// TwinCAT 3 PLC project Haltbergholz
// ProgramVersion: 3.1.4026.19
// libraries:
//   Tc2_ModbusSrv, * (Beckhoff Automation GmbH)
//   Tc2_Standard, * (Beckhoff Automation GmbH)
//   Tc2_System, * (Beckhoff Automation GmbH)
//   Tc2_Utilities, * (Beckhoff Automation GmbH)
//   Tc3_EventLogger, * (Beckhoff Automation GmbH)
// project tree:
//   DUTs/ E_PhaseSelect.TcDUT, E_StorageChargeState.TcDUT
//   DUTs/FroniusModbusRegisterMapping/ ST_RegMapInverter.TcDUT, ST_RegMapMeter.TcDUT, ST_RegMapStorage.TcDUT
//   DUTs/GridOperatingData/ ST_OpDataInverter.TcDUT, ST_OpDataMeter.TcDUT, ST_OpDataStorage.TcDUT
//   DUTs/LoadControlData/ ST_CtrlDataPower.TcDUT, ST_CtrlDataSetpoint.TcDUT
//   DUTs/Properties/ ST_SchmittTriggerProperties.TcDUT
//   / PlcTask.TcTTO
//   POUs/ FB_ModbusCon.TcPOU, FB_SchmittTrigger.TcPOU, F_MovingAverage.TcPOU, I_LoadCtrl.TcIO, MainCtrl.TcPOU
// real-time tasks:
//   TASK PlcTask: cycle T#10ms, priority 20, ADS port 350

CONFIGURATION Haltbergholz
    RESOURCE PLC ON TwinCAT3
        TASK PlcTask(INTERVAL := T#10ms, PRIORITY := 20);
        PROGRAM MainCtrl WITH PlcTask : MainCtrl;
    END_RESOURCE
END_CONFIGURATION

// ---- DUTs/E_PhaseSelect.TcDUT
{attribute 'qualified_only'}
{attribute 'strict'}
{attribute 'to_string'}
TYPE E_PhaseSelect :
(
	ALL := 0,
    L1,
    L2,
    L3
);
END_TYPE

// ---- DUTs/E_StorageChargeState.TcDUT
{attribute 'qualified_only'}
{attribute 'strict'}
{attribute 'to_string'}
TYPE E_StorageChargeState :
(
	off := 1,
    empty := 2,
    discharging := 3,
    charging := 4,
    full := 5,
    holding := 6,
    testing := 7
) WORD;
END_TYPE

// ---- DUTs/FroniusModbusRegisterMapping/ST_RegMapInverter.TcDUT
TYPE ST_RegMapInverter :
STRUCT
    // Register 40072
    nCurrentTotal: WORD;
    // Register 40073
    nCurrentL1: WORD;
    // Register 40074
    nCurrentL2: WORD;
    // Register 40075
    nCurrentL3: WORD;
    // Register 40076
    nSfCurrent: WORD;
    // Register 40077
    nVoltageL1L2: WORD;
    // Register 40078
    nVoltageL2L3: WORD;
    // Register 40079
    nVoltageL3L1: WORD;
    // Register 40080
    nVoltageL1N: WORD;
    // Register 40081
    nVoltageL2N: WORD;
    // Register 40082
    nVoltageL3N: WORD;
    // Register 40083
    nSfVoltage: WORD;
    // Register 40084
    nPower: WORD;
    // Register 40085
    nSfPower: WORD;
    // Register 40086
    nFrequency: WORD;
    // Register 40087
    nSfFrequency: WORD;
END_STRUCT
END_TYPE

// ---- DUTs/FroniusModbusRegisterMapping/ST_RegMapMeter.TcDUT
TYPE ST_RegMapMeter :
STRUCT
    // Register 40072
    nCurrentTotal: WORD;
    // Register 40073
    nCurrentL1: WORD;
    // Register 40074
    nCurrentL2: WORD;
    // Register 40075
    nCurrentL3: WORD;
    // Register 40076
    nSfCurrent: WORD;
    // Register 40077
    nVoltageLN: WORD;
    // Register 40078
    nVoltageL1N: WORD;
    // Register 40079
    nVoltageL2N: WORD;
    // Register 40080
    nVoltageL3N: WORD;
    // Register 40081
    nVoltageLL: WORD;
    // Register 40082
    nVoltageL1L2: WORD;
    // Register 40083
    nVoltageL2L3: WORD;
    // Register 40084
    nVoltageL3L1: WORD;
    // Register 40085
    nSfVoltage: WORD;
    // Register 40086
    nFrequency: WORD;
    // Register 40087
    nSfFrequency: WORD;
    // Register 40088
    nPower: WORD;
    // Register 40089
    nPowerL1: WORD;
    // Register 40090
    nPowerL2: WORD;
    // Register 40091
    nPowerL3: WORD;
    // Register 40092
    nSfPower: WORD;
END_STRUCT
END_TYPE

// ---- DUTs/FroniusModbusRegisterMapping/ST_RegMapStorage.TcDUT
TYPE ST_RegMapStorage :
STRUCT
    // Register 40352
    nStateOfCharge: WORD;
    // Register 40353
    nStorageAvailable: WORD;
    // Register 40354
    nVoltageInternal: WORD;
    // Register 40355
    nState: E_StorageChargeState;
    // Register 40366, fixed to -2
    nSfStateOfCharge: WORD := INT_TO_UINT(-2);
END_STRUCT
END_TYPE

// ---- DUTs/GridOperatingData/ST_OpDataInverter.TcDUT
TYPE ST_OpDataInverter :
STRUCT
    // Operating data refreshed in this cycle
    bOpDataIsUpdated: BOOL;
    // Current Phase L1 [A]
    fCurrentL1: REAL;
    // Current Phase L2 [A]
    fCurrentL2: REAL;
    // Current Phase L3 [A]
    fCurrentL3: REAL;
    // Voltage between Phase L1 and L2 [V]
    fVoltageL1L2: REAL;
    // Voltage between Phase L2 and L3 [V]
    fVoltageL2L3: REAL;
    // Voltage between Phase L3 and L1 [V]
    fVoltageL3L1: REAL;
    // Voltage between Phase L1 and N [V]
    fVoltageL1N: REAL;
    // Voltage between Phase L2 and N [V]
    fVoltageL2N: REAL;
    // Voltage between Phase L3 and N [V]
    fVoltageL3N: REAL;
    // Total Real Power [W]
    fPower: REAL;
    // Frequency [Hz]
    fFrequency: REAL;
END_STRUCT
END_TYPE

// ---- DUTs/GridOperatingData/ST_OpDataMeter.TcDUT
TYPE ST_OpDataMeter :
STRUCT
    // Operating data refreshed in this cycle
    bOpDataIsUpdated: BOOL;
    // Current Phase L1 [A]
    fCurrentL1: REAL;
    // Current Phase L2 [A]
    fCurrentL2: REAL;
    // Current Phase L3 [A]
    fCurrentL3: REAL;
    // Voltage between Phase L1 and L2 [V]
    fVoltageL1L2: REAL;
    // Voltage between Phase L2 and L3 [V]
    fVoltageL2L3: REAL;
    // Voltage between Phase L3 and L1 [V]
    fVoltageL3L1: REAL;
    // Voltage between Phase L1 and N [V]
    fVoltageL1N: REAL;
    // Voltage between Phase L2 and N [V]
    fVoltageL2N: REAL;
    // Voltage between Phase L3 and N [V]
    fVoltageL3N: REAL;
    // Total Real Power [W]
    fPower: REAL;
    // Real Power of Phase L1 [W]
    fPowerL1: REAL;
    // Real Power of Phase L2 [W]
    fPowerL2: REAL;
    // Real Power of Phase L3 [W]
    fPowerL3: REAL;
    // Frequency [Hz]
    fFrequency: REAL;
END_STRUCT
END_TYPE

// ---- DUTs/GridOperatingData/ST_OpDataStorage.TcDUT
TYPE ST_OpDataStorage :
STRUCT
    // Operating data refreshed in this cycle
    bOpDataIsUpdated: BOOL;
    // Currently available energy as a percent of the capacity rating
    nStateOfCharge: INT;
    // Charge status of storage device
    eState: E_StorageChargeState;
END_STRUCT
END_TYPE

// ---- DUTs/LoadControlData/ST_CtrlDataPower.TcDUT
TYPE ST_CtrlDataPower :
STRUCT
    // Real Power of Phase L1 [W]
    fPowerL1: REAL;
    // Real Power of Phase L2 [W]
    fPowerL2: REAL;
    // Real Power of Phase L3 [W]
    fPowerL3: REAL;
END_STRUCT
END_TYPE

// ---- DUTs/LoadControlData/ST_CtrlDataSetpoint.TcDUT
TYPE ST_CtrlDataSetpoint :
STRUCT
    // Load setpoint for Phase L1 [0-255]
    nLoadSetpointL1: USINT;
    // Load setpoint for Phase L2 [0-255]
    nLoadSetpointL2: USINT;
    // Load setpoint for Phase L3 [0-255]
    nLoadSetpointL3: USINT;
END_STRUCT
END_TYPE

// ---- DUTs/Properties/ST_SchmittTriggerProperties.TcDUT
TYPE ST_SchmittTriggerProperties :
STRUCT
    // Number of oscillations (t < threashold) required to reverse output
    nLimitOscillations: INT;
    // Time threshold to switch output after falling edge of input
    tFallThreshold: TIME;
    // Time threshold to switch output after rising edge of input
    tRiseThreshold: TIME;
END_STRUCT
END_TYPE

// ---- POUs/I_LoadCtrl.TcIO
INTERFACE I_LoadCtrl

// True if load is ready to powered on
{attribute 'monitoring' := 'variable'}
PROPERTY bReady : BOOL
GET
END_GET
END_PROPERTY

// Show only events with minimum severety level
{attribute 'monitoring' := 'call'}
PROPERTY eTraceLevel: Global.TcEventSeverity
GET
END_GET
SET
END_SET
END_PROPERTY

// Release power up of load on selected phase
METHOD PowerDown : BOOL
VAR_INPUT
    ePhase: E_PhaseSelect := E_PhaseSelect.ALL;
END_VAR
END_METHOD

// Power down load on selected phase
METHOD PowerUp : BOOL
VAR_INPUT
    ePhase: E_PhaseSelect := E_PhaseSelect.ALL;
END_VAR
END_METHOD

// Request setpoint for poweroutput relative to stPowerMaximum
{attribute 'monitoring' := 'call'}
PROPERTY stLoadSetpoint : REFERENCE TO ST_CtrlDataSetpoint
GET
END_GET
SET
END_SET
END_PROPERTY

// Actual power used from load
{attribute 'monitoring' := 'variable'}
PROPERTY stPowerActual : REFERENCE TO ST_CtrlDataPower
GET
END_GET
END_PROPERTY

// Minimum power on lowest setpoint
{attribute 'monitoring' := 'variable'}
PROPERTY stPowerMaximum : REFERENCE TO ST_CtrlDataPower
GET
END_GET
END_PROPERTY

// Maxmimum power on highest setpoint
{attribute 'monitoring' := 'variable'}
PROPERTY stPowerMinimum : REFERENCE TO ST_CtrlDataPower
GET
END_GET
END_PROPERTY

END_INTERFACE

// ---- POUs/MainCtrl.TcPOU
PROGRAM MainCtrl
VAR
    fbReadOpData: FB_ModbusCon := (
                    sInverterIPAddr := '127.0.0.1',
                    nInverterTCPPort := 5502,
                    nInverterUnitID := 16#01,
                    nMeterUnitID := 16#C8,
                    tConnectionTimeout := T#10S,
                    tConnectionCoolDown := T#10S);

    // Load control 1
    ipLoad1: I_LoadCtrl;

    // Battery is charging
    fbStorageIsCharging: FB_SchmittTrigger;

    // Temporary Power of Phase L1 values used for moving average 
    aMeterHistoryPowerL1: ARRAY[1..nSamplesMovingAverage] OF REAL;
    nMeterHistoryCursorPowerL1: INT;
    // Temporary Power of Phase L2 values used for moving average 
    aMeterHistoryPowerL2: ARRAY[1..nSamplesMovingAverage] OF REAL;
    nMeterHistoryCursorPowerL2: INT;
    // Temporary Power of Phase L3 values used for moving average 
    aMeterHistoryPowerL3: ARRAY[1..nSamplesMovingAverage] OF REAL;
    nMeterHistoryCursorPowerL3: INT;

    // Actual power feed to grid (>0: feed to grid, <0: draw from grid)
    stSurplusPower: ST_CtrlDataPower;
    // Surplus available at Phase L1
    fbSurplusAvailableL1: FB_SchmittTrigger;
    // Surplus available at Phase L2
    fbSurplusAvailableL2: FB_SchmittTrigger;
    // Surplus available at Phase L3
    fbSurplusAvailableL3: FB_SchmittTrigger;
END_VAR
VAR PERSISTENT
    // Battery state of charge is high
    nStorageStateOfChargeHigh: INT := 75;
    // Schmitt trigger configuration for battery charging state while battery state of charge low
    stStorageIsChargingTriggerPropertiesLow: ST_SchmittTriggerProperties := (
                                        nLimitOscillations := 3,
                                        tFallThreshold := T#5M,
                                        tRiseThreshold := T#2M);
    // Schmitt trigger configuration for battery charging state while battery state of charge high
    stStorageIsChargingTriggerPropertiesHigh: ST_SchmittTriggerProperties := (
                                        nLimitOscillations := 3,
                                        tFallThreshold := T#2M,
                                        tRiseThreshold := T#2M);
    // Schmitt trigger configuration for surplus power active while battery state of charge low
    stSurplusPowerTriggerPropertiesLow: ST_SchmittTriggerProperties := (
                                        nLimitOscillations := 3,
                                        tFallThreshold := T#5M,
                                        tRiseThreshold := T#1M);
    // Schmitt trigger configuration for surplus power active while battery state of charge high
    stSurplusPowerTriggerPropertiesHigh: ST_SchmittTriggerProperties := (
                                        nLimitOscillations := 3,
                                        tFallThreshold := T#50M,
                                        tRiseThreshold := T#1M);
    // Minimum amount of power feed to grid must be exceeded to show as surplus (>=0W)
    stSurplusPowerMinimum: ST_CtrlDataPower := (
                                        fPowerL1 := 20,
                                        fPowerL2 := 20,
                                        fPowerL3 := 20);
END_VAR
VAR CONSTANT
    // Number of samples for moving average calculation
    nSamplesMovingAverage: INT := 3;
END_VAR

// Fetch measurement data
fbReadOpData();

IF NOT fbReadOpData.bReady THEN
    fbReadOpData.bEnable := FALSE;
    RETURN;
ELSE
    fbReadOpData.bEnable := TRUE;
END_IF

// Battery measurement data is updated
IF fbReadOpData.stStorage.bOpDataIsUpdated THEN
    IF fbReadOpData.stStorage.nStateOfCharge > nStorageStateOfChargeHigh THEN
        fbStorageIsCharging.nLimitOscillations := stStorageIsChargingTriggerPropertiesLow.nLimitOscillations;
        fbStorageIsCharging.tFallThreshold := stStorageIsChargingTriggerPropertiesLow.tFallThreshold;
        fbStorageIsCharging.tRiseThreshold := stStorageIsChargingTriggerPropertiesLow.tRiseThreshold;
    ELSE
        fbStorageIsCharging.nLimitOscillations := stStorageIsChargingTriggerPropertiesHigh.nLimitOscillations;
        fbStorageIsCharging.tFallThreshold := stStorageIsChargingTriggerPropertiesHigh.tFallThreshold;
        fbStorageIsCharging.tRiseThreshold := stStorageIsChargingTriggerPropertiesHigh.tRiseThreshold;
    END_IF

    // Detect change on battery charging state
    fbStorageIsCharging.bIn := fbReadOpData.stStorage.eState = E_StorageChargeState.charging;
END_IF

fbStorageIsCharging();

// Meter measurement data is updated
IF fbReadOpData.stMeter.bOpDataIsUpdated THEN
    // Get moving average of power measured at meter and reverse sign (>0: feed to grid, <0: draw from grid)
    stSurplusPower.fPowerL1 := F_MovingAverage(fIn := fbReadOpData.stMeter.fPowerL1, aHisotry := aMeterHistoryPowerL1, nCursor := nMeterHistoryCursorPowerL1) * -1;
    stSurplusPower.fPowerL2 := F_MovingAverage(fIn := fbReadOpData.stMeter.fPowerL2, aHisotry := aMeterHistoryPowerL2, nCursor := nMeterHistoryCursorPowerL2) * -1;
    stSurplusPower.fPowerL3 := F_MovingAverage(fIn := fbReadOpData.stMeter.fPowerL3, aHisotry := aMeterHistoryPowerL3, nCursor := nMeterHistoryCursorPowerL3) * -1;

    // Add the actual power used of the loads to surplus (further calculations without used power of all load)
    IncludeLoadToSurplus(ipLoad := ipLoad1);

    // Generate setpoint for each load
    GenerateSetpoint(ipLoad := ipLoad1);

    // Detect change between power feed and draw to grid
    fbSurplusAvailableL1.bIn := stSurplusPower.fPowerL1 >= stSurplusPowerMinimum.fPowerL1;
    fbSurplusAvailableL2.bIn := stSurplusPower.fPowerL2 >= stSurplusPowerMinimum.fPowerL2;
    fbSurplusAvailableL3.bIn := stSurplusPower.fPowerL3 >= stSurplusPowerMinimum.fPowerL3;
END_IF

// Set properties of surplus available trigger based on battery charging state
IF fbStorageIsCharging.bOut THEN
    fbSurplusAvailableL1.nLimitOscillations := stSurplusPowerTriggerPropertiesLow.nLimitOscillations;
    fbSurplusAvailableL1.tFallThreshold := stSurplusPowerTriggerPropertiesLow.tFallThreshold;
    fbSurplusAvailableL1.tRiseThreshold := stSurplusPowerTriggerPropertiesLow.tRiseThreshold;
    fbSurplusAvailableL2.nLimitOscillations := stSurplusPowerTriggerPropertiesLow.nLimitOscillations;
    fbSurplusAvailableL2.tFallThreshold := stSurplusPowerTriggerPropertiesLow.tFallThreshold;
    fbSurplusAvailableL2.tRiseThreshold := stSurplusPowerTriggerPropertiesLow.tRiseThreshold;
    fbSurplusAvailableL3.nLimitOscillations := stSurplusPowerTriggerPropertiesLow.nLimitOscillations;
    fbSurplusAvailableL3.tFallThreshold := stSurplusPowerTriggerPropertiesLow.tFallThreshold;
    fbSurplusAvailableL3.tRiseThreshold := stSurplusPowerTriggerPropertiesLow.tRiseThreshold;
ELSE
    fbSurplusAvailableL1.nLimitOscillations := stSurplusPowerTriggerPropertiesHigh.nLimitOscillations;
    fbSurplusAvailableL1.tFallThreshold := stSurplusPowerTriggerPropertiesHigh.tFallThreshold;
    fbSurplusAvailableL1.tRiseThreshold := stSurplusPowerTriggerPropertiesHigh.tRiseThreshold;
    fbSurplusAvailableL2.nLimitOscillations := stSurplusPowerTriggerPropertiesHigh.nLimitOscillations;
    fbSurplusAvailableL2.tFallThreshold := stSurplusPowerTriggerPropertiesHigh.tFallThreshold;
    fbSurplusAvailableL2.tRiseThreshold := stSurplusPowerTriggerPropertiesHigh.tRiseThreshold;
    fbSurplusAvailableL3.nLimitOscillations := stSurplusPowerTriggerPropertiesHigh.nLimitOscillations;
    fbSurplusAvailableL3.tFallThreshold := stSurplusPowerTriggerPropertiesHigh.tFallThreshold;
    fbSurplusAvailableL3.tRiseThreshold := stSurplusPowerTriggerPropertiesHigh.tRiseThreshold;
END_IF

fbSurplusAvailableL1();
fbSurplusAvailableL2();
fbSurplusAvailableL3();

// Enable / Disable Load 1 on phase 1
IF fbSurplusAvailableL1.bOut AND ipLoad1.bReady THEN
    ipLoad1.PowerUp(ePhase := E_PhaseSelect.L1);
ELSE
    ipLoad1.PowerDown(ePhase := E_PhaseSelect.L1);
END_IF

// Enable / Disable Load 1 on phase 2
IF fbSurplusAvailableL2.bOut AND ipLoad1.bReady THEN
    ipLoad1.PowerUp(ePhase := E_PhaseSelect.L2);
ELSE
    ipLoad1.PowerDown(ePhase := E_PhaseSelect.L2);
END_IF

// Enable / Disable Load 1 on phase 3
IF fbSurplusAvailableL3.bOut AND ipLoad1.bReady THEN
    ipLoad1.PowerUp(ePhase := E_PhaseSelect.L3);
ELSE
    ipLoad1.PowerDown(ePhase := E_PhaseSelect.L3);
END_IF

// Generate and append setpoint of each phase to stLoadSetpoint of interface based on stPowerMaximum of interface and the current stSurplusPower 
METHOD PRIVATE GenerateSetpoint
VAR_INPUT
    // Interface of load control
    ipLoad: REFERENCE TO I_LoadCtrl;
END_VAR
IF ipLoad.stPowerMaximum.fPowerL1 <= 0 THEN
    ipLoad.stLoadSetpoint.nLoadSetpointL1 := 0;
ELSE
    ipLoad.stLoadSetpoint.nLoadSetpointL1 := REAL_TO_USINT(LIMIT(0, stSurplusPower.fPowerL1 / ipLoad.stPowerMaximum.fPowerL1, 1) * 255);
END_IF

IF ipLoad.stPowerMaximum.fPowerL2 <= 0 THEN
    ipLoad.stLoadSetpoint.nLoadSetpointL2 := 0;
ELSE
    ipLoad.stLoadSetpoint.nLoadSetpointL2 := REAL_TO_USINT(LIMIT(0, stSurplusPower.fPowerL2 / ipLoad.stPowerMaximum.fPowerL2, 1) * 255);
END_IF

IF ipLoad.stPowerMaximum.fPowerL3 <= 0 THEN
    ipLoad.stLoadSetpoint.nLoadSetpointL3 := 0;
ELSE
    ipLoad.stLoadSetpoint.nLoadSetpointL3 := REAL_TO_USINT(LIMIT(0, stSurplusPower.fPowerL3 / ipLoad.stPowerMaximum.fPowerL3, 1) * 255);
END_IF
END_METHOD

// Add the actual power used of the load to surplus
METHOD PRIVATE IncludeLoadToSurplus
VAR_INPUT
    // Interface of load control
    ipLoad: REFERENCE TO I_LoadCtrl;
END_VAR
stSurplusPower.fPowerL1 := stSurplusPower.fPowerL1 + ipLoad.stPowerActual.fPowerL1;
stSurplusPower.fPowerL2 := stSurplusPower.fPowerL2 + ipLoad.stPowerActual.fPowerL2;
stSurplusPower.fPowerL3 := stSurplusPower.fPowerL3 + ipLoad.stPowerActual.fPowerL3;
END_METHOD

END_PROGRAM

// ---- POUs/FB_ModbusCon.TcPOU
FUNCTION_BLOCK FB_ModbusCon
VAR_INPUT
    bEnable: BOOL;
END_VAR
VAR_OUTPUT
    // Operating data from inverter
    stInverter: ST_OpDataInverter;
    // Operating data from meter
    stMeter: ST_OpDataMeter;
    // Operating data from storage
    stStorage: ST_OpDataStorage;
    // Connection is ready and not locked out
    bReady: BOOL;
END_VAR
VAR
    // IP address of the target device
    {attribute 'hide'}
    _sInverterIPAddr: STRING;
    // Port number of the target device
    {attribute 'hide'}
    _nInverterTCPPort: UINT;
    // Modbus RTU ID of inverter, value must be 16#FF if addressed directly via TCP/IP
    {attribute 'hide'}
    _nInverterUnitID: BYTE;
    // Modbus RTU ID of meter, value must be 16#FF if addressed directly via TCP/IP
    {attribute 'hide'}
    _nMeterUnitID: BYTE;
    // Timeout that may not be exceeded by execution of the ADS command
    {attribute 'hide'}
    _tConnectionTimeout: TIME;
    // Timeout between modbus commands sent to target device
    {attribute 'hide'}
    _tConnectionCoolDown: TIME;

    // Modbus connection to read registers
    fbReadRegister: FB_MBReadRegs;
    // Connection cooldown timeout between requests
    fbConnectionCoolDown: TOF;

    // Register data of inverter
    stInverterRegisterData: ST_RegMapInverter;
    // Register data of meter
    stMeterRegisterData: ST_RegMapMeter;
    // Register data of storage
    stStorageRegisterData: ST_RegMapStorage;

    // Number of current tried countermeasures after modbus connection error
    nConnectionCountermeasure: INT;
    // Number of current tried countermeasures after modbus request error regarding inverter
    nInverterCountermeasure: INT;
    // Number of current tried countermeasures after modbus request error regarding meter
    nMeterCountermeasure: INT;
    // Number of current tried countermeasures after modbus request error regarding storage
    nStorageCountermeasure: INT;

    // Current state of modbus read registers
    eReadState: (WAIT_FOR_ENABLE, PREPARE_READ_REGS, EXECUTE_READ_REGS, WAIT_READ_REGS_FEEDBACK, ASSIGN_VALUES, SELECT_NEXT_SUBSYTEM, CON_COOL_DOWN, CON_LOCKOUT);
    // Select subsystem for request to prevent parallel requests
    eCurrentSubsystem: (INVERTER, METER, STORAGE);

    // Show only events with minimum severety level
    {attribute 'hide'}
    _eTraceLevel: TcEventSeverity := TcEventSeverity.Warning;

    fbAlarmMbConnectionError: FB_TcAlarm;
    fbAlarmMbFunctionInverterError: FB_TcAlarm;
    fbAlarmMbFunctionMeterError: FB_TcAlarm;
    fbAlarmMbFunctionStorageError: FB_TcAlarm;
    fbAlarmMbConnectionLocked: FB_TcAlarm;
    fbMessageMbOpDataIsUpdated: FB_TcMessage;
    fbMessageMbUncatchedError: FB_TcMessage;
    fbMessageMbReceivedBytesMismatch: FB_TcMessage;
END_VAR
VAR CONSTANT
    // Number of output registers used by stInverterRegisterData
    nInverterRegQuantity: WORD := 16;
    // Start address of the output register used by stInverterRegisterData
    nInverterMBStartAddr: WORD := 40071;
    // Number of output registers used by stMeterRegisterData
    nMeterRegQuantity: WORD := 21;
    // Start address of the output register used by stMeterRegisterData
    nMeterMBStartAddr: WORD := 40071;
    // Number of output registers used by stStorageRegisterData
    nStorageRegQuantity: WORD := 4;
    // Start address of the output register used by stStorageRegisterData
    nStorageMBStartAddr: WORD := 40351;
    // Number of attempted countermeasures before connection lockout (connection error)
    nConnectionCmBeforeLockout: INT := 5;
    // Number of attempted countermeasures before connection lockout (subsystem error)
    nSubsystemCmBeforeLockout: INT := 2;
END_VAR

fbReadRegister(sIPAddr := sInverterIPAddr, nTCPPort := nInverterTCPPort, tTimeout := tConnectionTimeout);
fbConnectionCoolDown();

// Set ready state
bReady := eReadState <> CON_LOCKOUT;

// Default operating data has not been updated this cycle
stInverter.bOpDataIsUpdated := FALSE;
stMeter.bOpDataIsUpdated := FALSE;
stStorage.bOpDataIsUpdated := FALSE;

// State machine
CASE eReadState OF
    WAIT_FOR_ENABLE:
        IF bEnable AND fbConnectionCoolDown.Q THEN
            eReadState := CON_COOL_DOWN;
        ELSIF bEnable THEN
            eReadState := PREPARE_READ_REGS;
        END_IF

    PREPARE_READ_REGS:
        CASE eCurrentSubsystem OF
            INVERTER:
                fbReadRegister.nUnitID := nInverterUnitID;
                fbReadRegister.nQuantity := nInverterRegQuantity;
                fbReadRegister.nMBAddr := nInverterMBStartAddr;
                fbReadRegister.cbLength := SIZEOF(stInverterRegisterData);
                fbReadRegister.pDestAddr := ADR(stInverterRegisterData);

            METER:
                fbReadRegister.nUnitID := nMeterUnitID;
                fbReadRegister.nQuantity := nMeterRegQuantity;
                fbReadRegister.nMBAddr := nMeterMBStartAddr;
                fbReadRegister.cbLength := SIZEOF(stMeterRegisterData);
                fbReadRegister.pDestAddr := ADR(stMeterRegisterData);

            STORAGE:
                fbReadRegister.nUnitID := nInverterUnitID;
                fbReadRegister.nQuantity := nStorageRegQuantity;
                fbReadRegister.nMBAddr := nStorageMBStartAddr;
                fbReadRegister.cbLength := SIZEOF(stStorageRegisterData) - 2;
                fbReadRegister.pDestAddr := ADR(stStorageRegisterData);
        END_CASE

        eReadState := EXECUTE_READ_REGS;

    EXECUTE_READ_REGS:
        fbReadRegister.bExecute := TRUE;
        fbConnectionCoolDown.IN := TRUE;
        eReadState := WAIT_READ_REGS_FEEDBACK;

    WAIT_READ_REGS_FEEDBACK:
        fbReadRegister.bExecute := FALSE;
        IF NOT fbReadRegister.bBusy THEN
            fbConnectionCoolDown.IN := FALSE;
            ConnectionErrorHandler();

            IF ConnectionLockoutIsActive() THEN
                // Lockout modbus connection
                eReadState := CON_LOCKOUT;
            ELSIF fbReadRegister.cbLength <> fbReadRegister.cbRead THEN
                // Send message M_MbReceivedBytesMismatch
                IF fbMessageMbReceivedBytesMismatch.eSeverity >= eTraceLevel THEN
                    fbMessageMbReceivedBytesMismatch.ipArguments.Clear();
                    fbMessageMbReceivedBytesMismatch.ipArguments.AddBool(value := eCurrentSubsystem = INVERTER);
                    fbMessageMbReceivedBytesMismatch.ipArguments.AddBool(value := eCurrentSubsystem = METER);
                    fbMessageMbReceivedBytesMismatch.ipArguments.AddBool(value := eCurrentSubsystem = STORAGE);
                    fbMessageMbReceivedBytesMismatch.Send();
                END_IF
                // Skip assigning values to output variable
                eReadState := SELECT_NEXT_SUBSYTEM;
            ELSE
                eReadState := ASSIGN_VALUES;
            END_IF
        END_IF

    ASSIGN_VALUES:
        CASE eCurrentSubsystem OF
            INVERTER:
                stInverter.bOpDataIsUpdated := TRUE;
                stInverter.fCurrentL1 := Scale(stInverterRegisterData.nCurrentL1, stInverterRegisterData.nSfCurrent);
                stInverter.fCurrentL2 := Scale(stInverterRegisterData.nCurrentL2, stInverterRegisterData.nSfCurrent);
                stInverter.fCurrentL3 := Scale(stInverterRegisterData.nCurrentL3, stInverterRegisterData.nSfCurrent);
                stInverter.fVoltageL1L2 := Scale(stInverterRegisterData.nVoltageL1L2, stInverterRegisterData.nSfVoltage);
                stInverter.fVoltageL2L3 := Scale(stInverterRegisterData.nVoltageL2L3, stInverterRegisterData.nSfVoltage);
                stInverter.fVoltageL3L1 := Scale(stInverterRegisterData.nVoltageL3L1, stInverterRegisterData.nSfVoltage);
                stInverter.fVoltageL1N := Scale(stInverterRegisterData.nVoltageL1N, stInverterRegisterData.nSfVoltage);
                stInverter.fVoltageL2N := Scale(stInverterRegisterData.nVoltageL2N, stInverterRegisterData.nSfVoltage);
                stInverter.fVoltageL3N := Scale(stInverterRegisterData.nVoltageL3N, stInverterRegisterData.nSfVoltage);
                stInverter.fPower := Scale(stInverterRegisterData.nPower, stInverterRegisterData.nSfPower);
                stInverter.fFrequency := Scale(stInverterRegisterData.nFrequency, stInverterRegisterData.nSfFrequency);

            METER:
                stMeter.bOpDataIsUpdated := TRUE;
                stMeter.fCurrentL1 := Scale(stMeterRegisterData.nCurrentL1, stMeterRegisterData.nSfCurrent);
                stMeter.fCurrentL2 := Scale(stMeterRegisterData.nCurrentL2, stMeterRegisterData.nSfCurrent);
                stMeter.fCurrentL3 := Scale(stMeterRegisterData.nCurrentL3, stMeterRegisterData.nSfCurrent);
                stMeter.fVoltageL1L2 := Scale(stMeterRegisterData.nVoltageL1L2, stMeterRegisterData.nSfVoltage);
                stMeter.fVoltageL2L3 := Scale(stMeterRegisterData.nVoltageL2L3, stMeterRegisterData.nSfVoltage);
                stMeter.fVoltageL3L1 := Scale(stMeterRegisterData.nVoltageL3L1, stMeterRegisterData.nSfVoltage);
                stMeter.fVoltageL1N := Scale(stMeterRegisterData.nVoltageL1N, stMeterRegisterData.nSfVoltage);
                stMeter.fVoltageL2N := Scale(stMeterRegisterData.nVoltageL2N, stMeterRegisterData.nSfVoltage);
                stMeter.fVoltageL3N := Scale(stMeterRegisterData.nVoltageL3N, stMeterRegisterData.nSfVoltage);
                stMeter.fPower := Scale(stMeterRegisterData.nPower, stMeterRegisterData.nSfPower);
                stMeter.fPowerL1 := Scale(stMeterRegisterData.nPowerL1, stMeterRegisterData.nSfPower);
                stMeter.fPowerL2 := Scale(stMeterRegisterData.nPowerL2, stMeterRegisterData.nSfPower);
                stMeter.fPowerL3 := Scale(stMeterRegisterData.nPowerL3, stMeterRegisterData.nSfPower);
                stMeter.fFrequency := Scale(stMeterRegisterData.nFrequency, stMeterRegisterData.nSfFrequency);

            STORAGE:
                stStorage.bOpDataIsUpdated := TRUE;
                stStorage.nStateOfCharge := REAL_TO_INT(Scale(stStorageRegisterData.nStateOfCharge, stStorageRegisterData.nSfStateOfCharge));
                stStorage.eState := stStorageRegisterData.nState;
        END_CASE
        eReadState := SELECT_NEXT_SUBSYTEM;

        // Send message M_MbOpDataIsUpdated
        IF fbMessageMbOpDataIsUpdated.eSeverity >= eTraceLevel THEN
            fbMessageMbOpDataIsUpdated.ipArguments.Clear();
            fbMessageMbOpDataIsUpdated.ipArguments.AddBool(value := stInverter.bOpDataIsUpdated);
            fbMessageMbOpDataIsUpdated.ipArguments.AddBool(value := stMeter.bOpDataIsUpdated);
            fbMessageMbOpDataIsUpdated.ipArguments.AddBool(value := stStorage.bOpDataIsUpdated);
            fbMessageMbOpDataIsUpdated.Send();
        END_IF

    SELECT_NEXT_SUBSYTEM:
        CASE eCurrentSubsystem OF
            INVERTER:
                eCurrentSubsystem := METER;

            METER:
                eCurrentSubsystem := STORAGE;

            STORAGE:
                eCurrentSubsystem := INVERTER;

            ELSE
                eCurrentSubsystem := INVERTER;
        END_CASE
        eReadState := CON_COOL_DOWN;

    CON_COOL_DOWN:
        IF NOT bEnable THEN
            eReadState := WAIT_FOR_ENABLE;
        END_IF

        IF NOT fbConnectionCoolDown.Q THEN
            eReadState := PREPARE_READ_REGS;
        END_IF

    CON_LOCKOUT:
        (* Perform reset using Reset() function *)
END_CASE

METHOD PRIVATE ConnectionErrorHandler
IF ConnectionLockoutIsActive() THEN
    RETURN;
END_IF

IF fbReadRegister.bError THEN
    // Apply countermeasure if ADS error occured
    CASE fbReadRegister.nErrId OF
        16#8001, // Modbus function not implemented
        16#8002, // Invalid address or length
        16#8003, // Invalid parameters: incorrect number of registers
        16#8004: // Modbus server error
            CASE eCurrentSubsystem OF
                INVERTER:
                    nInverterCountermeasure := nInverterCountermeasure + 1;
                METER:
                    nMeterCountermeasure := nMeterCountermeasure + 1;
                STORAGE:
                    nStorageCountermeasure := nStorageCountermeasure + 1;
            END_CASE
            

        Global.E_TcSystemEventClass.TCPSendError, // TCP send error
        Tc2_System.E_AdsErr.CLIENT_SYNCTIMEOUT:   // Remote terminal is not responding in the specified ADS timeout
            nConnectionCountermeasure := nConnectionCountermeasure + 1;
            fbConnectionCoolDown.PT := tConnectionCoolDown + tConnectionCoolDown * LREAL_TO_INT(EXPT(nConnectionCountermeasure, 2));

        ELSE
            // Send message M_MbUncatchedError
            IF fbMessageMbUncatchedError.eSeverity >= eTraceLevel THEN
                fbMessageMbUncatchedError.ipArguments.Clear();
                fbMessageMbUncatchedError.ipArguments.AddUDInt(value := fbReadRegister.nErrId);
                fbMessageMbUncatchedError.Send();
            END_IF
    END_CASE

ELSE
    // Defer possibly still active countermeasure
    nInverterCountermeasure := 0;
    nMeterCountermeasure := 0;
    nStorageCountermeasure := 0;
    nConnectionCountermeasure := 0;

    // Reset connection cooldown timeout
    fbConnectionCoolDown.PT := tConnectionCoolDown;
END_IF

IF nConnectionCountermeasure > 0 AND fbAlarmMbConnectionError.eSeverity >= eTraceLevel AND NOT fbAlarmMbConnectionError.bRaised THEN
    // Raise alarm F_MbConnectionError
    fbAlarmMbConnectionError.ipArguments.AddUDInt(value := fbReadRegister.nErrId);
    fbAlarmMbConnectionError.Raise();
ELSIF nConnectionCountermeasure = 0 AND fbAlarmMbConnectionError.bRaised THEN
    // Clear alarm F_MbConnectionError
    fbAlarmMbConnectionError.ipArguments.Clear();
    fbAlarmMbConnectionError.Clear();
END_IF

IF nInverterCountermeasure > 0 AND fbAlarmMbFunctionInverterError.eSeverity >= eTraceLevel AND NOT fbAlarmMbFunctionInverterError.bRaised THEN
    // Raise alarm F_MbFunctionInverterError
    fbAlarmMbFunctionInverterError.ipArguments.AddUDInt(value := fbReadRegister.nErrId);
    fbAlarmMbFunctionInverterError.Raise();
ELSIF nInverterCountermeasure = 0 AND fbAlarmMbFunctionInverterError.bRaised THEN
    // Clear alarm F_MbFunctionInverterError
    fbAlarmMbFunctionInverterError.ipArguments.Clear();
    fbAlarmMbFunctionInverterError.Clear();
END_IF

IF nMeterCountermeasure > 0 AND fbAlarmMbFunctionMeterError.eSeverity >= eTraceLevel AND NOT fbAlarmMbFunctionMeterError.bRaised THEN
    // Raise alarm F_MbFunctionMeterError
    fbAlarmMbFunctionMeterError.ipArguments.AddUDInt(value := fbReadRegister.nErrId);
    fbAlarmMbFunctionMeterError.Raise();
ELSIF nMeterCountermeasure = 0 AND fbAlarmMbFunctionMeterError.bRaised THEN
    // Clear alarm F_MbFunctionMeterError
    fbAlarmMbFunctionMeterError.ipArguments.Clear();
    fbAlarmMbFunctionMeterError.Clear();
END_IF

IF nStorageCountermeasure > 0 AND fbAlarmMbFunctionStorageError.eSeverity >= eTraceLevel AND NOT fbAlarmMbFunctionStorageError.bRaised THEN
    // Raise alarm F_MbFunctionStorageError
    fbAlarmMbFunctionStorageError.ipArguments.AddUDInt(value := fbReadRegister.nErrId);
    fbAlarmMbFunctionStorageError.Raise();
ELSIF nStorageCountermeasure = 0 AND fbAlarmMbFunctionStorageError.bRaised THEN
    // Clear alarm F_MbFunctionStorageError
    fbAlarmMbFunctionStorageError.ipArguments.Clear();
    fbAlarmMbFunctionStorageError.Clear();
END_IF
END_METHOD

METHOD PRIVATE ConnectionLockoutIsActive : BOOL
// Default to false, no lockout active
ConnectionLockoutIsActive := FALSE;

// Return if already in locked state
IF eReadState = CON_LOCKOUT THEN
    ConnectionLockoutIsActive := TRUE;
    RETURN;
END_IF

IF nConnectionCountermeasure > nConnectionCmBeforeLockout THEN
    ConnectionLockoutIsActive := TRUE;
    // Add reference to F_MbConnectionError as argument to F_MbConnectionLocked
    IF fbAlarmMbConnectionLocked.eSeverity >= eTraceLevel AND NOT fbAlarmMbConnectionLocked.bRaised THEN
        fbAlarmMbConnectionLocked.ipArguments.AddEventReferenceId(nEventId := fbAlarmMbConnectionError.nEventId);
    END_IF
END_IF

if nInverterCountermeasure > nSubsystemCmBeforeLockout THEN
    ConnectionLockoutIsActive := TRUE;
    // Add reference to F_MbFunctionInverterError as argument to F_MbConnectionLocked
    IF fbAlarmMbConnectionLocked.eSeverity >= eTraceLevel AND NOT fbAlarmMbConnectionLocked.bRaised THEN
        fbAlarmMbConnectionLocked.ipArguments.AddEventReferenceId(nEventId := fbAlarmMbFunctionInverterError.nEventId);
    END_IF
END_IF

if nMeterCountermeasure > nSubsystemCmBeforeLockout THEN
    ConnectionLockoutIsActive := TRUE;
    // Add reference to F_MbFunctionMeterError as argument to F_MbConnectionLocked
    IF fbAlarmMbConnectionLocked.eSeverity >= eTraceLevel AND NOT fbAlarmMbConnectionLocked.bRaised THEN
        fbAlarmMbConnectionLocked.ipArguments.AddEventReferenceId(nEventId := fbAlarmMbFunctionMeterError.nEventId);
    END_IF
END_IF

if nStorageCountermeasure > nSubsystemCmBeforeLockout THEN
    ConnectionLockoutIsActive := TRUE;
    // Add reference to F_MbFunctionStorageError as argument to F_MbConnectionLocked
    IF fbAlarmMbConnectionLocked.eSeverity >= eTraceLevel AND NOT fbAlarmMbConnectionLocked.bRaised THEN
        fbAlarmMbConnectionLocked.ipArguments.AddEventReferenceId(nEventId := fbAlarmMbFunctionStorageError.nEventId);
    END_IF
END_IF

IF ConnectionLockoutIsActive AND fbAlarmMbConnectionLocked.eSeverity >= eTraceLevel AND NOT fbAlarmMbConnectionLocked.bRaised THEN
    // Raise alarm F_MbConnectionLocked
    fbAlarmMbConnectionLocked.Raise();
END_IF
END_METHOD

// Show only events with minimum severety level
{attribute 'monitoring' := 'call'}
PROPERTY eTraceLevel : Global.TcEventSeverity
GET
eTraceLevel := _eTraceLevel;
END_GET
SET
_eTraceLevel := eTraceLevel;
END_SET
END_PROPERTY

METHOD FB_Init: BOOL
VAR_INPUT
    // TRUE: the retain variables are initialized (reset warm / reset cold)
    bInitRetains: BOOL;
    // TRUE: the instance will be copied to the copy code afterward (online change)
    bInCopyCode: BOOL; 
END_VAR
// Create alarm/message instances for the event logger
IF NOT bInCopyCode THEN
    fbAlarmMbConnectionError.CreateEx(stEventEntry := TC_EVENTS.MainControllerEventClass.F_MbConnectionError, bWithConfirmation := FALSE);
    fbAlarmMbFunctionInverterError.CreateEx(stEventEntry := TC_EVENTS.MainControllerEventClass.F_MbFunctionInverterError, bWithConfirmation := FALSE);
    fbAlarmMbFunctionMeterError.CreateEx(stEventEntry := TC_EVENTS.MainControllerEventClass.F_MbFunctionMeterError, bWithConfirmation := FALSE);
    fbAlarmMbFunctionStorageError.CreateEx(stEventEntry := TC_EVENTS.MainControllerEventClass.F_MbFunctionStorageError, bWithConfirmation := FALSE);
    fbAlarmMbConnectionLocked.CreateEx(stEventEntry := TC_EVENTS.MainControllerEventClass.F_MbConnectionLocked, bWithConfirmation := FALSE);
    fbMessageMbOpDataIsUpdated.CreateEx(stEventEntry := TC_EVENTS.MainControllerEventClass.M_MbOpDataIsUpdated);
    fbMessageMbUncatchedError.CreateEx(stEventEntry := TC_EVENTS.MainControllerEventClass.M_MbUncatchedError);
    fbMessageMbReceivedBytesMismatch.CreateEx(stEventEntry := TC_EVENTS.MainControllerEventClass.M_MbReceivedBytesMismatch);
END_IF
END_METHOD

// IP address of the target device
{attribute 'monitoring' := 'variable'}
PROPERTY nInverterTCPPort : UINT
GET
nInverterTCPPort := _nInverterTCPPort;
END_GET
SET
_nInverterTCPPort := nInverterTCPPort;
END_SET
END_PROPERTY

// Modbus RTU ID of inverter, value must be 16#FF if addressed directly via TCP/IP
{attribute 'monitoring' := 'variable'}
PROPERTY nInverterUnitID : BYTE
GET
nInverterUnitID := _nInverterUnitID;
END_GET
SET
_nInverterUnitID := nInverterUnitID;
END_SET
END_PROPERTY

// Modbus RTU ID of meter, value must be 16#FF if addressed directly via TCP/IP
{attribute 'monitoring' := 'variable'}
PROPERTY nMeterUnitID : BYTE
GET
nMeterUnitID := _nMeterUnitID;
END_GET
SET
_nMeterUnitID := nMeterUnitID;
END_SET
END_PROPERTY

METHOD PUBLIC Reset
nInverterCountermeasure := 0;
nMeterCountermeasure := 0;
nStorageCountermeasure := 0;
nConnectionCountermeasure := 0;

eReadState := WAIT_FOR_ENABLE;

// Clear alarm F_MbConnectionLocked
fbAlarmMbConnectionLocked.Clear();
fbAlarmMbConnectionLocked.ipArguments.Clear();
END_METHOD

METHOD PRIVATE Scale : REAL
VAR_INPUT
    nValue: WORD;
    nScaleFactor: WORD;
END_VAR
Scale := nValue * LREAL_TO_REAL(EXPT(10, UINT_TO_INT(nScaleFactor)));
END_METHOD

// IP address of the target device
{attribute 'monitoring' := 'variable'}
PROPERTY sInverterIPAddr : STRING
GET
sInverterIPAddr := _sInverterIPAddr;
END_GET
SET
_sInverterIPAddr := sInverterIPAddr;
END_SET
END_PROPERTY

// Timeout between modbus commands sent to target device
{attribute 'monitoring' := 'call'}
PROPERTY tConnectionCoolDown : TIME
GET
tConnectionCoolDown := _tConnectionCoolDown;
END_GET
SET
_tConnectionCoolDown := tConnectionCoolDown;

// Apply connection cooldown timeout if no counter measure is active
IF nConnectionCountermeasure = 0 AND nInverterCountermeasure = 0 AND nMeterCountermeasure = 0 AND nStorageCountermeasure = 0 THEN
    fbConnectionCoolDown.PT := tConnectionCoolDown;
END_IF
END_SET
END_PROPERTY

// Timeout that may not be exceeded by execution of the ADS command
{attribute 'monitoring' := 'call'}
PROPERTY tConnectionTimeout : TIME
GET
tConnectionTimeout := _tConnectionTimeout;
END_GET
SET
_tConnectionTimeout := tConnectionTimeout;
END_SET
END_PROPERTY

END_FUNCTION_BLOCK

// ---- POUs/FB_SchmittTrigger.TcPOU
FUNCTION_BLOCK FB_SchmittTrigger
VAR_INPUT
    bIn: BOOL;
END_VAR
VAR_OUTPUT
    bOut: BOOL;
END_VAR
VAR
    // Number of oscillations for output switch before threshold reached
    {attribute 'hide'}
    _nLimitOscillations: INT;

    // Last input stored
    bInLast: BOOL;
    // Count of oscollations (falling / rising edge depending on bOut) while one threshold counter is active
    nOscillations: INT;
    // Time threshold to switch output after falling edge of input
    fbFallThreshold: TON;
    // Time threshold to switch output after rising edge of input
    fbRiseThreshold: TON;
END_VAR

fbFallThreshold();
fbRiseThreshold();

IF bIn <> bInLast THEN
    // Input falling edge
    IF NOT bIn THEN
        fbFallThreshold.IN := TRUE;
        fbRiseThreshold.IN := FALSE;

        // Increase oscillation counter if falling edge threashold timer has not reached tFallThreshold
        IF bOut AND NOT fbFallThreshold.Q THEN
            nOscillations := nOscillations + 1;
        END_IF

    // Input rising edge
    ELSIF bIn THEN
        fbFallThreshold.IN := FALSE;
        fbRiseThreshold.IN := TRUE;

        // Increase oscillation counter if rising edge threashold timer has not reached tRiseThreshold
        IF NOT bOut AND NOT fbRiseThreshold.Q THEN
            nOscillations := nOscillations + 1;
        END_IF
    END_IF

    // Store last input on change
    bInLast := bIn;
END_IF

// Set output bit, reset threshold timer, reset oscillation counter
IF fbFallThreshold.Q OR nLimitOscillations > 0 AND nOscillations >= nLimitOscillations AND bOut THEN
    bOut := FALSE;
    fbFallThreshold.IN := FALSE;
    nOscillations := 0;
ELSIF fbRiseThreshold.Q OR nLimitOscillations > 0 AND nOscillations >= nLimitOscillations AND NOT bOut THEN
    bOut := TRUE;
    fbRiseThreshold.IN := FALSE;
    nOscillations := 0;
END_IF

// Number of oscillations (t < threashold) required to reverse output
{attribute 'monitoring' := 'call'}
PROPERTY nLimitOscillations : INT
GET
nLimitOscillations := _nLimitOscillations;
END_GET
SET
_nLimitOscillations := nLimitOscillations;
END_SET
END_PROPERTY

// Time threshold to switch output after falling edge of input
{attribute 'monitoring' := 'call'}
PROPERTY tFallThreshold : TIME
GET
tFallThreshold := fbFallThreshold.PT;
END_GET
SET
fbFallThreshold.PT := tFallThreshold;
END_SET
END_PROPERTY

// Time threshold to switch output after rising edge of input
{attribute 'monitoring' := 'call'}
PROPERTY tRiseThreshold : TIME
GET
tRiseThreshold := fbRiseThreshold.PT;
END_GET
SET
fbRiseThreshold.PT := tRiseThreshold;
END_SET
END_PROPERTY

END_FUNCTION_BLOCK

// ---- POUs/F_MovingAverage.TcPOU
FUNCTION F_MovingAverage : REAL
VAR_INPUT
    fIn: REAL;
END_VAR
VAR_IN_OUT
    aHisotry: ARRAY[*] OF REAL;
    nCursor: INT;
END_VAR
VAR
    nLower: INT;
    nUpper: INT;
    n: DINT;
    fSum: REAL;
END_VAR

nLower := DINT_TO_INT(LOWER_BOUND(aHisotry, 1));
nUpper := DINT_TO_INT(UPPER_BOUND(aHisotry, 1));

// Append new value to array
aHisotry[nCursor] := fIn;
// Move cursor for next input
IF nCursor < nUpper - nLower + 1 THEN
    nCursor := nCursor + 1;
ELSE
    nCursor := nLower;
END_IF

// Calculate average
n := nLower;
WHILE n <= nUpper DO
    fSum := fSum + aHisotry[n];
    n := n + 1;
END_WHILE

F_MovingAverage := fSum / (nUpper - nLower + 1);

END_FUNCTION
